FUNCTION_BLOCK FB_Diag
VAR_OUTPUT
	Alarm: BOOL;
	Vorwarn: BOOL;
	Meld: BOOL;
END_VAR

Alarm := TRUE;
Vorwarn := TRUE;
Meld := TRUE;

END_FUNCTION_BLOCK

(* stored: Version 1.1.0.1, ProductVersion 3.1.0.12
   POU FB_Diag: Id {a88242f6-fb2d-4fb1-b417-5c69a9a55e74} *)
